FUNCTION_BLOCK UDINT_AUDI_AX_SEL (* binary selection *)
  (* Standard: 61499-2; Description: Copyright (c) 2026 HR Agrartechnik GmbH This program and the accompanying materials are made available under the terms of the Eclipse Public License 2.0 which is available at https://www.eclipse.org/legal/epl-2.0/ SPDX-License-Identifier: EPL-2.0 *)
  (* Version 1.0, 2026-04-19, Franz Höpfinger, HR Agrartechnik GmbH, initial API and implementation *)
  PACKAGE adapter::iec61131::selection;
  IMPORT eclipse4diac::core::TypeHash;
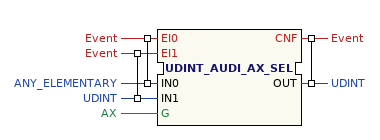
  EVENT_INPUT
    EI0 WITH IN0; (* Set IN0 *)
    EI1 WITH IN1; (* Set IN1 *)
  END_EVENT
  EVENT_OUTPUT
    CNF WITH OUT; (* Confirmation of Requested Service *)
  END_EVENT
  VAR_INPUT
    IN0 : ANY_ELEMENTARY; (* Selectable input variable *)
    IN1 : UDINT; (* Selectable input variable *)
  END_VAR
  VAR_OUTPUT
    OUT : UDINT; (* Selected input *)
  END_VAR
  SOCKETS
    G : adapter::types::unidirectional::AX; (* Selelctor *)
  END_SOCKETS
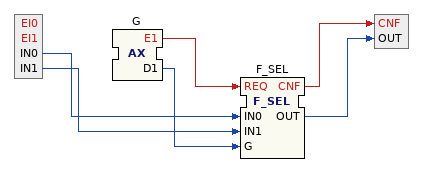
  FBS
    F_SEL : iec61131::selection::F_SEL;
  END_FBS
  EVENT_CONNECTIONS
    F_SEL.CNF TO CNF;
    G.E1 TO F_SEL.REQ;
  END_CONNECTIONS
  DATA_CONNECTIONS
    IN0 TO F_SEL.IN0;
    IN1 TO F_SEL.IN1;
    F_SEL.OUT TO OUT;
    G.D1 TO F_SEL.G;
  END_CONNECTIONS
END_FUNCTION_BLOCK
